// TIA Portal V19 export
TYPE "C402_VAR_SBO_TYPIC"
   STRUCT
      BEZ_STS { ExternalAccessible := 'False'; ExternalVisible := 'False'; ExternalWritable := 'False'} : USInt;   // Status van de beweging van de afsluitboom
      POS_STS { ExternalAccessible := 'False'; ExternalVisible := 'False'; ExternalWritable := 'False'} : USInt;   // Status van de positie van de afsluitboom
      BMO { ExternalAccessible := 'False'; ExternalVisible := 'False'; ExternalWritable := 'False'} : USInt;   // Bedieningsmode
      BST { ExternalAccessible := 'False'; ExternalVisible := 'False'; ExternalWritable := 'False'} : USInt;   // Bestuurbaarheid
   END_STRUCT;
END_TYPE
